// TIA Portal V17 export
// export: Created 2026-07-06T15:32:59.266637Z, ExportSetting WithDefaults, DisplayName Totally Integrated Automation Portal, DisplayVersion V17, DisplayName TIA Portal Openness, DisplayVersion V17, DisplayName TIA Portal Version Control Interface, DisplayVersion V17, DisplayName STEP 7 Professional, DisplayVersion V17, DisplayName STEP 7 Safety, DisplayVersion V17, DisplayName WinCC Professional, DisplayVersion V17
ORGANIZATION_BLOCK "Main"   // OB1, LAD, ProgramCycle
TITLE = "Main Program Sweep (Cycle)"
{ S7_Optimized_Access := 'TRUE' }
VERSION : 0.1
// stored: AutoNumber true, IsIECCheckEnabled false, SetENOAutomatically false
   VAR_INPUT
      Initial_Call : Bool;   // Initial call of this OB
      Remanence : Bool;   // =True, if remanent data are available
   END_VAR
BEGIN

REGION Network 1
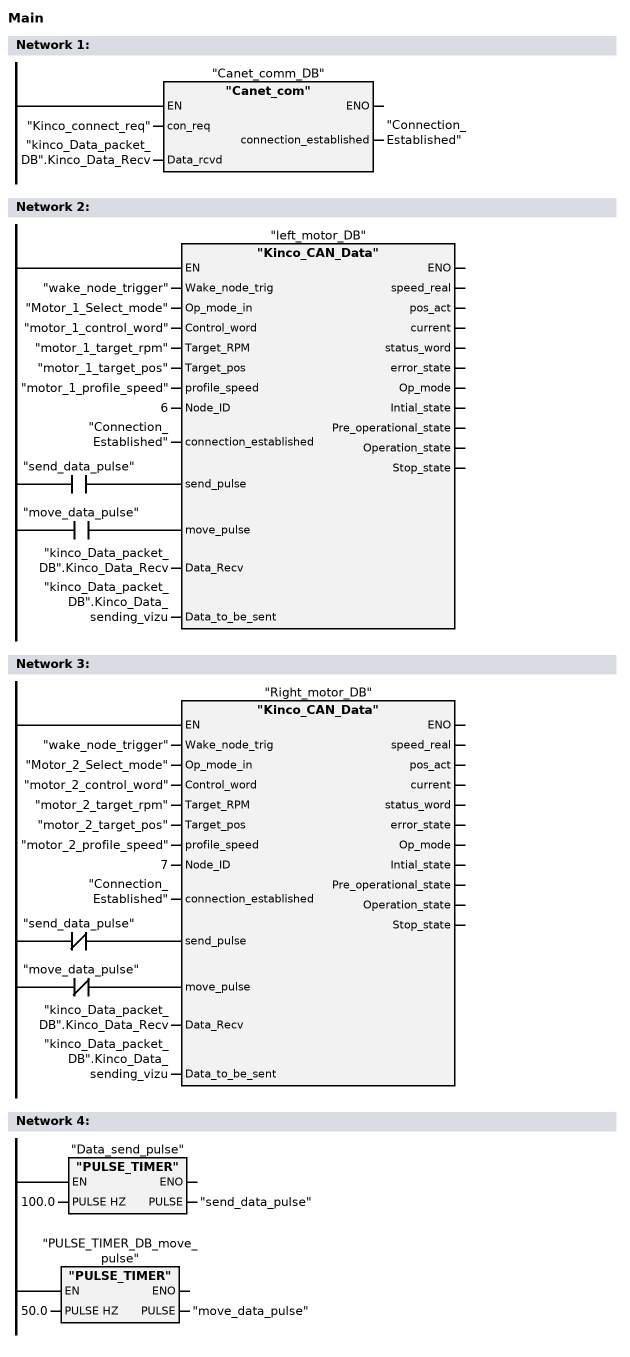
   RUNG wire#powerrail
      "Canet_comm_DB"(con_req := "Kinco_connect_req", Data_rcvd := "kinco_Data_packet_DB".Kinco_Data_Recv, connection_established => "Connection_Established")
   END_RUNG
   // the same network as SCL:
   "Canet_comm_DB"(con_req := "Kinco_connect_req",   // "Canet_com"
                   Data_rcvd := "kinco_Data_packet_DB".Kinco_Data_Recv,
                   connection_established => "Connection_Established");
END_REGION

REGION Network 2
   RUNG wire#powerrail
      "left_motor_DB"(send_pulse := wire#w1, move_pulse := wire#w2, Wake_node_trig := "wake_node_trigger", Op_mode_in := "Motor_1_Select_mode", Control_word := "motor_1_control_word", Target_RPM := "motor_1_target_rpm", Target_pos := "motor_1_target_pos", profile_speed := "motor_1_profile_speed", Node_ID := 6, connection_established := "Connection_Established", Data_Recv := "kinco_Data_packet_DB".Kinco_Data_Recv, Data_to_be_sent := "kinco_Data_packet_DB".Kinco_Data_sending_vizu, speed_real =>, pos_act =>, current =>, status_word =>, error_state =>, Op_mode =>, Intial_state =>, Pre_operational_state =>, Operation_state =>, Stop_state =>)
   END_RUNG
   RUNG wire#powerrail
      Contact( "send_data_pulse" )
   END_RUNG wire#w1
   RUNG wire#powerrail
      Contact( "move_data_pulse" )
   END_RUNG wire#w2
   // the same network as SCL:
   "left_motor_DB"(Wake_node_trig := "wake_node_trigger",   // "Kinco_CAN_Data"
                   Op_mode_in := "Motor_1_Select_mode",
                   Control_word := "motor_1_control_word",
                   Target_RPM := "motor_1_target_rpm",
                   Target_pos := "motor_1_target_pos",
                   profile_speed := "motor_1_profile_speed",
                   Node_ID := 6,
                   connection_established := "Connection_Established",
                   send_pulse := "send_data_pulse",
                   move_pulse := "move_data_pulse",
                   Data_Recv := "kinco_Data_packet_DB".Kinco_Data_Recv,
                   Data_to_be_sent := "kinco_Data_packet_DB".Kinco_Data_sending_vizu);
END_REGION

REGION Network 3
   RUNG wire#powerrail
      "Right_motor_DB"(send_pulse := wire#w1, move_pulse := wire#w2, Wake_node_trig := "wake_node_trigger", Op_mode_in := "Motor_2_Select_mode", Control_word := "motor_2_control_word", Target_RPM := "motor_2_target_rpm", Target_pos := "motor_2_target_pos", profile_speed := "motor_2_profile_speed", Node_ID := 7, connection_established := "Connection_Established", Data_Recv := "kinco_Data_packet_DB".Kinco_Data_Recv, Data_to_be_sent := "kinco_Data_packet_DB".Kinco_Data_sending_vizu, speed_real =>, pos_act =>, current =>, status_word =>, error_state =>, Op_mode =>, Intial_state =>, Pre_operational_state =>, Operation_state =>, Stop_state =>)
   END_RUNG
   RUNG wire#powerrail
      I_Contact( "send_data_pulse" )
   END_RUNG wire#w1
   RUNG wire#powerrail
      I_Contact( "move_data_pulse" )
   END_RUNG wire#w2
   // the same network as SCL:
   "Right_motor_DB"(Wake_node_trig := "wake_node_trigger",   // "Kinco_CAN_Data"
                    Op_mode_in := "Motor_2_Select_mode",
                    Control_word := "motor_2_control_word",
                    Target_RPM := "motor_2_target_rpm",
                    Target_pos := "motor_2_target_pos",
                    profile_speed := "motor_2_profile_speed",
                    Node_ID := 7,
                    connection_established := "Connection_Established",
                    send_pulse := NOT "send_data_pulse",
                    move_pulse := NOT "move_data_pulse",
                    Data_Recv := "kinco_Data_packet_DB".Kinco_Data_Recv,
                    Data_to_be_sent := "kinco_Data_packet_DB".Kinco_Data_sending_vizu);
END_REGION

REGION Network 4
   RUNG wire#powerrail
      "Data_send_pulse"("PULSE HZ" := 100.0, PULSE => "send_data_pulse")
   END_RUNG
   RUNG wire#powerrail
      "PULSE_TIMER_DB_move_pulse"("PULSE HZ" := 50.0, PULSE => "move_data_pulse")
   END_RUNG
   // the same network as SCL:
   "Data_send_pulse"("PULSE HZ" := 100.0, PULSE => "send_data_pulse");   // "PULSE_TIMER"
   "PULSE_TIMER_DB_move_pulse"("PULSE HZ" := 50.0, PULSE => "move_data_pulse");   // "PULSE_TIMER"
END_REGION
END_ORGANIZATION_BLOCK
